    clear_socket_buffer("1")
    clear_socket_buffer("2")
    clear_socket_buffer("3")
    clear_socket_buffer("4")
    # end: URCap Program Node
    # begin: URCap Program Node
    #   Source: Robotiq_Grippers, 1.6.0.4, Robotiq Inc.
    #   Type: Gripper
    gripper_1_used = True
    if (connectivity_checked[0] != 1):
      if not(rq_set_sid(9, "1")):
        popup("Gripper 1 must be connected to run this program.", "No connection", False, True, True)
      end
      connectivity_checked[0] = 1
    end
    if (status_checked[0] != 1):
      if not(rq_is_gripper_activated("1")):
        popup("Gripper 1 is not activated. Go to Installation tab > Gripper to activate it and run the program again.", "Not activated", False, True, True)
      end
      status_checked[0] = 1
    end
    rq_set_pos_spd_for(128, 255, 255, "1")
    rq_go_to("1")
    rq_wait("1")
    gripper_1_selected = True
    gripper_2_selected = False
    gripper_3_selected = False
    gripper_4_selected = False
    gripper_1_used = False
    gripper_2_used = False
    gripper_3_used = False
    gripper_4_used = False
    # end: URCap Program Node
    movej(get_inverse_kin(home_p, qnear=home_q), a=1.3962634015954636, v=1.0471975511965976)
    movej(get_inverse_kin(ra_b1_wp_p, qnear=ra_b1_wp_q), a=1.3962634015954636, v=1.0471975511965976)
    movej(get_inverse_kin(ra_b1_at_p, qnear=ra_b1_at_q), a=1.3962634015954636, v=1.0471975511965976)
    # begin: URCap Program Node
    #   Source: Robotiq_Grippers, 1.6.0.4, Robotiq Inc.
    #   Type: Gripper
    gripper_1_used = True
    if (connectivity_checked[0] != 1):
      if not(rq_set_sid(9, "1")):
        popup("Gripper 1 must be connected to run this program.", "No connection", False, True, True)
      end
      connectivity_checked[0] = 1
    end
    if (status_checked[0] != 1):
      if not(rq_is_gripper_activated("1")):
        popup("Gripper 1 is not activated. Go to Installation tab > Gripper to activate it and run the program again.", "Not activated", False, True, True)
      end
      status_checked[0] = 1
    end
    rq_set_pos_spd_for(255, 255, 255, "1")
    rq_go_to("1")
    rq_wait("1")
    gripper_1_selected = True
    gripper_2_selected = False
    gripper_3_selected = False
    gripper_4_selected = False
    gripper_1_used = False
    gripper_2_used = False
    gripper_3_used = False
    gripper_4_used = False
    # end: URCap Program Node
    movej(get_inverse_kin(ra_b1_wp_p, qnear=ra_b1_wp_q), a=1.3962634015954636, v=1.0471975511965976)
    movej(get_inverse_kin(h_ra_b1_wp_p, qnear=h_ra_b1_wp_q), a=1.3962634015954636, v=1.0471975511965976)
    movej(get_inverse_kin(h_ra_b1_at_p, qnear=h_ra_b1_at_q), a=1.3962634015954636, v=1.0471975511965976)
    # begin: URCap Program Node
    #   Source: Robotiq_Grippers, 1.6.0.4, Robotiq Inc.
    #   Type: Gripper
    gripper_1_used = True
    if (connectivity_checked[0] != 1):
      if not(rq_set_sid(9, "1")):
        popup("Gripper 1 must be connected to run this program.", "No connection", False, True, True)
      end
      connectivity_checked[0] = 1
    end
    if (status_checked[0] != 1):
      if not(rq_is_gripper_activated("1")):
        popup("Gripper 1 is not activated. Go to Installation tab > Gripper to activate it and run the program again.", "Not activated", False, True, True)
      end
      status_checked[0] = 1
    end
    rq_set_pos_spd_for(128, 255, 255, "1")
    rq_go_to("1")
    rq_wait("1")
    gripper_1_selected = True
    gripper_2_selected = False
    gripper_3_selected = False
    gripper_4_selected = False
    gripper_1_used = False
    gripper_2_used = False
    gripper_3_used = False
    gripper_4_used = False
    # end: URCap Program Node
    movej(get_inverse_kin(h_ra_b1_wp_p, qnear=h_ra_b1_wp_q), a=1.3962634015954636, v=1.0471975511965976)
    movej(get_inverse_kin(ra_b2_wp_p, qnear=ra_b2_wp_q), a=1.3962634015954636, v=1.0471975511965976)
    movej(get_inverse_kin(ra_b2_at_p, qnear=ra_b2_at_q), a=1.3962634015954636, v=1.0471975511965976)
    # begin: URCap Program Node
    #   Source: Robotiq_Grippers, 1.6.0.4, Robotiq Inc.
    #   Type: Gripper
    gripper_1_used = True
    if (connectivity_checked[0] != 1):
      if not(rq_set_sid(9, "1")):
        popup("Gripper 1 must be connected to run this program.", "No connection", False, True, True)
      end
      connectivity_checked[0] = 1
    end
    if (status_checked[0] != 1):
      if not(rq_is_gripper_activated("1")):
        popup("Gripper 1 is not activated. Go to Installation tab > Gripper to activate it and run the program again.", "Not activated", False, True, True)
      end
      status_checked[0] = 1
    end
    rq_set_pos_spd_for(255, 255, 255, "1")
    rq_go_to("1")
    rq_wait("1")
    gripper_1_selected = True
    gripper_2_selected = False
    gripper_3_selected = False
    gripper_4_selected = False
    gripper_1_used = False
    gripper_2_used = False
    gripper_3_used = False
    gripper_4_used = False
    # end: URCap Program Node
    movej(get_inverse_kin(ra_b2_wp_p, qnear=ra_b2_wp_q), a=1.3962634015954636, v=1.0471975511965976)
    movej(get_inverse_kin(h_ra_b2_wp_p, qnear=h_ra_b2_wp_q), a=1.3962634015954636, v=1.0471975511965976)
    movej(get_inverse_kin(h_ra_b2_at_p, qnear=h_ra_b2_at_q), a=1.3962634015954636, v=1.0471975511965976)
    # begin: URCap Program Node
    #   Source: Robotiq_Grippers, 1.6.0.4, Robotiq Inc.
    #   Type: Gripper
    gripper_1_used = True
    if (connectivity_checked[0] != 1):
      if not(rq_set_sid(9, "1")):
        popup("Gripper 1 must be connected to run this program.", "No connection", False, True, True)
      end
      connectivity_checked[0] = 1
    end
    if (status_checked[0] != 1):
      if not(rq_is_gripper_activated("1")):
        popup("Gripper 1 is not activated. Go to Installation tab > Gripper to activate it and run the program again.", "Not activated", False, True, True)
      end
      status_checked[0] = 1
    end
    rq_set_pos_spd_for(128, 255, 255, "1")
    rq_go_to("1")
    rq_wait("1")
    gripper_1_selected = True
    gripper_2_selected = False
    gripper_3_selected = False
    gripper_4_selected = False
    gripper_1_used = False
    gripper_2_used = False
    gripper_3_used = False
    gripper_4_used = False
    # end: URCap Program Node
    movej(get_inverse_kin(h_ra_b2_wp_p, qnear=h_ra_b2_wp_q), a=1.3962634015954636, v=1.0471975511965976)
    movej(get_inverse_kin(home_p, qnear=home_q), a=1.3962634015954636, v=1.0471975511965976)
  end
  def reciprocal_p1_2():
    # begin: URCap Program Node
    #   Source: Robotiq_Grippers, 1.6.0.4, Robotiq Inc.
    #   Type: Gripper Activate

    rq_init_comm_if_connected(9, "1")
    rq_init_comm_if_connected(2, "2")
    rq_init_comm_if_connected(3, "3")
    rq_init_comm_if_connected(4, "4")

    reset_and_activate = False

    rq_activate_all_grippers(False)

    clear_socket_buffer("1")
    clear_socket_buffer("2")
    clear_socket_buffer("3")
    clear_socket_buffer("4")
    # end: URCap Program Node
    # begin: URCap Program Node
    #   Source: Robotiq_Grippers, 1.6.0.4, Robotiq Inc.
    #   Type: Gripper
    gripper_1_used = True
    if (connectivity_checked[0] != 1):
      if not(rq_set_sid(9, "1")):
        popup("Gripper 1 must be connected to run this program.", "No connection", False, True, True)
      end
      connectivity_checked[0] = 1
    end
    if (status_checked[0] != 1):
      if not(rq_is_gripper_activated("1")):
        popup("Gripper 1 is not activated. Go to Installation tab > Gripper to activate it and run the program again.", "Not activated", False, True, True)
      end
      status_checked[0] = 1
    end
    rq_set_pos_spd_for(128, 255, 255, "1")
    rq_go_to("1")
    rq_wait("1")
    gripper_1_selected = True
    gripper_2_selected = False
    gripper_3_selected = False
    gripper_4_selected = False
    gripper_1_used = False
    gripper_2_used = False
    gripper_3_used = False
    gripper_4_used = False
    # end: URCap Program Node
    movej(get_inverse_kin(home_p, qnear=home_q), a=1.3962634015954636, v=1.0471975511965976)
    movej(get_inverse_kin(m2_b1_wp_p, qnear=m2_b1_wp_q), a=1.3962634015954636, v=1.0471975511965976)
    movej(get_inverse_kin(m2_b1_at_p, qnear=m2_b1_at_q), a=1.3962634015954636, v=1.0471975511965976)
    # begin: URCap Program Node
    #   Source: Robotiq_Grippers, 1.6.0.4, Robotiq Inc.
    #   Type: Gripper
    gripper_1_used = True
    if (connectivity_checked[0] != 1):
      if not(rq_set_sid(9, "1")):
        popup("Gripper 1 must be connected to run this program.", "No connection", False, True, True)
      end
      connectivity_checked[0] = 1
    end
    if (status_checked[0] != 1):
      if not(rq_is_gripper_activated("1")):
        popup("Gripper 1 is not activated. Go to Installation tab > Gripper to activate it and run the program again.", "Not activated", False, True, True)
      end
      status_checked[0] = 1
    end
    rq_set_pos_spd_for(255, 255, 255, "1")
    rq_go_to("1")
    rq_wait("1")
    gripper_1_selected = True
    gripper_2_selected = False
    gripper_3_selected = False
    gripper_4_selected = False
    gripper_1_used = False
    gripper_2_used = False
    gripper_3_used = False
    gripper_4_used = False
    # end: URCap Program Node
    movej(get_inverse_kin(m2_b1_wp_p, qnear=m2_b1_wp_q), a=1.3962634015954636, v=1.0471975511965976)
    movej(get_inverse_kin(h_m2_b1_wp_p, qnear=h_m2_b1_wp_q), a=1.3962634015954636, v=1.0471975511965976)
    movej(get_inverse_kin(h_m2_b1_at_p, qnear=h_m2_b1_at_q), a=1.3962634015954636, v=1.0471975511965976)
    # begin: URCap Program Node
    #   Source: Robotiq_Grippers, 1.6.0.4, Robotiq Inc.
    #   Type: Gripper
    gripper_1_used = True
    if (connectivity_checked[0] != 1):
      if not(rq_set_sid(9, "1")):
        popup("Gripper 1 must be connected to run this program.", "No connection", False, True, True)
      end
      connectivity_checked[0] = 1
    end
    if (status_checked[0] != 1):
      if not(rq_is_gripper_activated("1")):
        popup("Gripper 1 is not activated. Go to Installation tab > Gripper to activate it and run the program again.", "Not activated", False, True, True)
      end
      status_checked[0] = 1
    end
    rq_set_pos_spd_for(128, 255, 255, "1")
    rq_go_to("1")
    rq_wait("1")
    gripper_1_selected = True
    gripper_2_selected = False
    gripper_3_selected = False
    gripper_4_selected = False
    gripper_1_used = False
    gripper_2_used = False
    gripper_3_used = False
    gripper_4_used = False
    # end: URCap Program Node
    movej(get_inverse_kin(h_m2_b1_wp_p, qnear=h_m2_b1_wp_q), a=1.3962634015954636, v=1.0471975511965976)
    movej(get_inverse_kin(home_p, qnear=home_q), a=1.3962634015954636, v=1.0471975511965976)
  end
  def reciprocal_p1_1():
    # begin: URCap Program Node
    #   Source: Robotiq_Grippers, 1.6.0.4, Robotiq Inc.
    #   Type: Gripper Activate

    rq_init_comm_if_connected(9, "1")
    rq_init_comm_if_connected(2, "2")
    rq_init_comm_if_connected(3, "3")
    rq_init_comm_if_connected(4, "4")

    reset_and_activate = False

    rq_activate_all_grippers(False)

    clear_socket_buffer("1")
    clear_socket_buffer("2")
    clear_socket_buffer("3")
    clear_socket_buffer("4")
    # end: URCap Program Node
    # begin: URCap Program Node
    #   Source: Robotiq_Grippers, 1.6.0.4, Robotiq Inc.
    #   Type: Gripper
    gripper_1_used = True
    if (connectivity_checked[0] != 1):
      if not(rq_set_sid(9, "1")):
        popup("Gripper 1 must be connected to run this program.", "No connection", False, True, True)
      end
      connectivity_checked[0] = 1
    end
    if (status_checked[0] != 1):
      if not(rq_is_gripper_activated("1")):
        popup("Gripper 1 is not activated. Go to Installation tab > Gripper to activate it and run the program again.", "Not activated", False, True, True)
      end
      status_checked[0] = 1
    end
    rq_set_pos_spd_for(128, 255, 255, "1")
    rq_go_to("1")
    rq_wait("1")
    gripper_1_selected = True
    gripper_2_selected = False
    gripper_3_selected = False
    gripper_4_selected = False
    gripper_1_used = False
    gripper_2_used = False
    gripper_3_used = False
    gripper_4_used = False
    # end: URCap Program Node
    movej(get_inverse_kin(home_p, qnear=home_q), a=1.3962634015954636, v=1.0471975511965976)
    movej(get_inverse_kin(b_b1_wp_p, qnear=b_b1_wp_q), a=1.3962634015954636, v=1.0471975511965976)
    movej(get_inverse_kin(b_b1_at_p, qnear=b_b1_at_q), a=1.3962634015954636, v=1.0471975511965976)
    # begin: URCap Program Node
    #   Source: Robotiq_Grippers, 1.6.0.4, Robotiq Inc.
    #   Type: Gripper
    gripper_1_used = True
    if (connectivity_checked[0] != 1):
      if not(rq_set_sid(9, "1")):
        popup("Gripper 1 must be connected to run this program.", "No connection", False, True, True)
      end
      connectivity_checked[0] = 1
    end
    if (status_checked[0] != 1):
      if not(rq_is_gripper_activated("1")):
        popup("Gripper 1 is not activated. Go to Installation tab > Gripper to activate it and run the program again.", "Not activated", False, True, True)
      end
      status_checked[0] = 1
    end
    rq_set_pos_spd_for(255, 255, 255, "1")
    rq_go_to("1")
    rq_wait("1")
    gripper_1_selected = True
    gripper_2_selected = False
    gripper_3_selected = False
    gripper_4_selected = False
    gripper_1_used = False
    gripper_2_used = False
    gripper_3_used = False
    gripper_4_used = False
    # end: URCap Program Node
    movej(get_inverse_kin(b_b1_wp_p, qnear=b_b1_wp_q), a=1.3962634015954636, v=1.0471975511965976)
    movej(get_inverse_kin(h_b_b1_wp_p, qnear=h_b_b1_wp_q), a=1.3962634015954636, v=1.0471975511965976)
    movej(get_inverse_kin(h_b_b1_at_p, qnear=h_b_b1_at_q), a=1.3962634015954636, v=1.0471975511965976)
    # begin: URCap Program Node
    #   Source: Robotiq_Grippers, 1.6.0.4, Robotiq Inc.
    #   Type: Gripper
    gripper_1_used = True
    if (connectivity_checked[0] != 1):
      if not(rq_set_sid(9, "1")):
        popup("Gripper 1 must be connected to run this program.", "No connection", False, True, True)
      end
      connectivity_checked[0] = 1
    end
    if (status_checked[0] != 1):
      if not(rq_is_gripper_activated("1")):
        popup("Gripper 1 is not activated. Go to Installation tab > Gripper to activate it and run the program again.", "Not activated", False, True, True)
      end
      status_checked[0] = 1
    end
    rq_set_pos_spd_for(128, 255, 255, "1")
    rq_go_to("1")
    rq_wait("1")
    gripper_1_selected = True
    gripper_2_selected = False
    gripper_3_selected = False
    gripper_4_selected = False
    gripper_1_used = False
    gripper_2_used = False
    gripper_3_used = False
    gripper_4_used = False
    # end: URCap Program Node
    movej(get_inverse_kin(h_b_b1_wp_p, qnear=h_b_b1_wp_q), a=1.3962634015954636, v=1.0471975511965976)
    movej(get_inverse_kin(b_b2_wp_p, qnear=b_b2_wp_q), a=1.3962634015954636, v=1.0471975511965976)
    movej(get_inverse_kin(b_b2_at_p, qnear=b_b2_at_q), a=1.3962634015954636, v=1.0471975511965976)
    # begin: URCap Program Node
    #   Source: Robotiq_Grippers, 1.6.0.4, Robotiq Inc.
    #   Type: Gripper
    gripper_1_used = True
    if (connectivity_checked[0] != 1):
      if not(rq_set_sid(9, "1")):
        popup("Gripper 1 must be connected to run this program.", "No connection", False, True, True)
      end
      connectivity_checked[0] = 1
    end
    if (status_checked[0] != 1):
      if not(rq_is_gripper_activated("1")):
        popup("Gripper 1 is not activated. Go to Installation tab > Gripper to activate it and run the program again.", "Not activated", False, True, True)
      end
      status_checked[0] = 1
    end
    rq_set_pos_spd_for(255, 255, 255, "1")
    rq_go_to("1")
    rq_wait("1")
    gripper_1_selected = True
    gripper_2_selected = False
    gripper_3_selected = False
    gripper_4_selected = False
    gripper_1_used = False
    gripper_2_used = False
    gripper_3_used = False
    gripper_4_used = False
    # end: URCap Program Node
    movej(get_inverse_kin(b_b2_wp_p, qnear=b_b2_wp_q), a=1.3962634015954636, v=1.0471975511965976)
    movej(get_inverse_kin(h_b_b2_wp_p, qnear=h_b_b2_wp_q), a=1.3962634015954636, v=1.0471975511965976)
    movej(get_inverse_kin(h_b_b2_at_p, qnear=h_b_b2_at_q), a=1.3962634015954636, v=1.0471975511965976)
    # begin: URCap Program Node
    #   Source: Robotiq_Grippers, 1.6.0.4, Robotiq Inc.
    #   Type: Gripper
    gripper_1_used = True
    if (connectivity_checked[0] != 1):
      if not(rq_set_sid(9, "1")):
        popup("Gripper 1 must be connected to run this program.", "No connection", False, True, True)
      end
      connectivity_checked[0] = 1
    end
    if (status_checked[0] != 1):
      if not(rq_is_gripper_activated("1")):
        popup("Gripper 1 is not activated. Go to Installation tab > Gripper to activate it and run the program again.", "Not activated", False, True, True)
      end
      status_checked[0] = 1
    end
    rq_set_pos_spd_for(128, 255, 255, "1")
    rq_go_to("1")
    rq_wait("1")
    gripper_1_selected = True
    gripper_2_selected = False
    gripper_3_selected = False
    gripper_4_selected = False
    gripper_1_used = False
    gripper_2_used = False
    gripper_3_used = False
    gripper_4_used = False
    # end: URCap Program Node
    movej(get_inverse_kin(h_b_b2_wp_p, qnear=h_b_b2_wp_q), a=1.3962634015954636, v=1.0471975511965976)
    movej(get_inverse_kin(home_p, qnear=home_q), a=1.3962634015954636, v=1.0471975511965976)
  end
  $ 1 "Robot Program"
  $ 2 "Call reciprocal_p1_1"
  reciprocal_p1_1()
  $ 3 "Popup"
  popup("interaction", "Message", False, False, blocking=True)
  $ 4 "Call reciprocal_p1_2"
  reciprocal_p1_2()
  $ 5 "Popup"
  popup("interaction", "Message", False, False, blocking=True)
  $ 6 "Call reciprocal_p1_3"
  reciprocal_p1_3()
  $ 7 "Popup"
  popup("interaction", "Message", False, False, blocking=True)
  $ 8 "Call reciprocal_p2_1"
  reciprocal_p2_1()
  $ 9 "Popup"
  popup("interaction", "Message", False, False, blocking=True)
  $ 10 "Call reciprocal_p2_2"
  reciprocal_p2_2()
  $ 11 "Popup"
  popup("interaction", "Message", False, False, blocking=True)
  $ 12 "Call reciprocal_p2_3"
  reciprocal_p2_3()
  $ 13 "Popup"
  popup("interaction", "Message", False, False, blocking=True)
  $ 14 "Call reciprocal_p3_1"
  reciprocal_p3_1()
  $ 15 "Popup"
  popup("interaction", "Message", False, False, blocking=True)
  $ 16 "Call reciprocal_p3_2"
  reciprocal_p3_2()
  $ 17 "Popup"
  popup("interaction", "Message", False, False, blocking=True)
  $ 18 "Call reciprocal_p3_3"
  reciprocal_p3_3()
end
